// Mitsubishi GX Works2 project: PLC 특수 기능 (PLS, PLF)   PLC: Q03UDV

PROGRAM MAIN
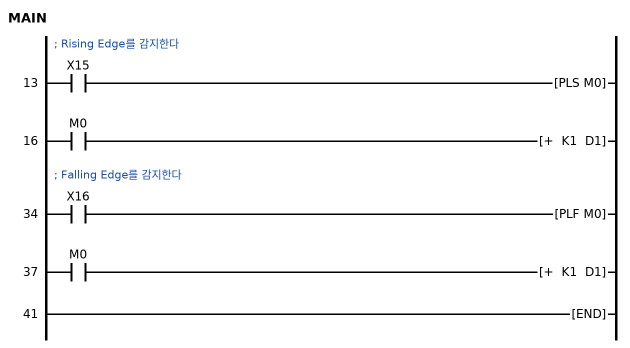
; Rising Edge를 감지한다
13    LD      X15
      PLS     M0
16    LD      M0
      +       K1 D1
; Falling Edge를 감지한다
34    LD      X16
      PLF     M0
37    LD      M0
      +       K1 D1
41    END
END_PROGRAM
